PROGRAM MAIN
VAR
	MyBoolean : BOOL;
	MyBoolean_2: BOOL;
	
	MyInt : INT;
	MyInt_2 : INT;
	
END_VAR



MyBoolean := TRUE;
MyInt:=3;

END_PROGRAM

(* stored: Version 1.1.0.1, ProductVersion 3.1.4024.11
   POU MAIN: Id {0829745f-6756-489d-bf06-f977de883d65}, SpecialFunc None *)
